Universal Robots URScript: move_path_1.script

def move_path_1():
  global _hidden_verificationVariable=0
  step_count_bb260f9f_b35d_4fa5_9196_51f97d34692a = 0.0
  thread Step_Counter_Thread_3f57fde8_be87_45f6_b73f_8ef8e3528eee():
    while (True):
      step_count_bb260f9f_b35d_4fa5_9196_51f97d34692a = step_count_bb260f9f_b35d_4fa5_9196_51f97d34692a + 1.0
      sync()
    end
  end
  run Step_Counter_Thread_3f57fde8_be87_45f6_b73f_8ef8e3528eee()
  set_gravity([0.0, 0.0, 9.82])
  set_standard_analog_input_domain(0, 1)
  set_standard_analog_input_domain(1, 1)
  set_tool_analog_input_domain(0, 1)
  set_tool_analog_input_domain(1, 1)
  set_analog_outputdomain(0, 0)
  set_analog_outputdomain(1, 0)
  set_input_actions_to_default()
  set_tcp(p[0.00855,-0.27152,0.102,1.2092,-1.2092,1.2092])
  set_target_payload(2.760000, [0.004000, -0.022000, 0.072000], [0.008360, 0.008360, 0.008360, 0.000000, 0.000000, 0.000000])
  set_safety_mode_transition_hardness(1)
  set_tool_communication(False, 115200, 0, 1, 1.5, 3.5)
  set_tool_output_mode(0)
  set_tool_digital_output_mode(0, 1)
  set_tool_digital_output_mode(1, 1)
  set_tool_voltage(0)
  global Plane_1=p[0.0,0.0,0.0,0.0,0.0,0.0]
  global Point_1=p[0.0,0.0,0.0,0.0,0.0,0.0]
  # begin: URCap Installation Node
  #   Source: MachineLogic for Universal Robots, 3.1.7, Vention Inc.
  #   Type: MachineLogic for Universal Robots
  def waitForResponse(expected_response_vention, cname_vention):
  response_vention = socket_read_string(cname_vention,timeout=15)
  while response_vention != expected_response_vention:
  sleep(0.01)
  response_vention = socket_read_string(cname_vention,timeout=15)
  end
  sleep(0.01)
  sync()
  end
  def sendString(string_vention, expected_response_vention, cname_vention):
  socket_send_string(str_cat(string_vention,";"), cname_vention)
  response_vention = socket_read_string(cname_vention,timeout=15)
  if(response_vention == "nAck"):
  popup("nAck received")
  end
  while response_vention != expected_response_vention:
  sleep(0.01)
  response_vention = socket_read_string(cname_vention,timeout=15)
  if(response_vention == "nAck"):
  popup("nAck received")
  end
  end
  sleep(0.01)
  sync()
  end
  def sendStringNAck(string_vention, expected_response_vention, cname_vention):
  socket_send_string(str_cat(string_vention,";"), cname_vention)
  response_vention = socket_read_string(cname_vention,timeout=15)
  if(response_vention == "nAck"):
  popup("nAck received")
  end
  while(response_vention != expected_response_vention and response_vention != "nAck"):
  sleep(0.01)
  response_vention = socket_read_string(cname_vention,timeout=15)
  if(response_vention == "nAck"):
  popup("nAck received",blocking=True)
  end
  end
  sleep(0.01)
  sync()
  end
  def sendStringWithTimeout(string_vention, expected_response_vention, cname_vention):
  socket_send_string(str_cat(string_vention,";"), cname_vention)
  response_vention = socket_read_string(cname_vention,timeout=10)
  if(response_vention == "nAck"):
  popup("nAck received"+string_vention)
  end
  sleep(0.01)
  sync()
  end
  def pollString(string_vention, expected_response_vention, cname_vention):
  socket_send_string(str_cat(string_vention,";"), cname_vention)
  response_vention = socket_read_string(cname_vention,timeout=15)
  if(response_vention == "nAck"):
  popup("nAck received")
  end
  while response_vention != expected_response_vention:
  sleep(1)
  socket_send_string(str_cat(string_vention,";"), cname_vention)
  response_vention = socket_read_string(cname_vention,timeout=15)
  if(response_vention == "nAck"):
  popup("nAck received")
  end
  end
  sleep(0.01)
  sync()
  end
  def sendVariable(var_vention, data_vention, expected_response_vention, cname_vention):
  socket_set_var(var_vention, data_vention, cname_vention)
  response_vention = socket_read_string(cname_vention,timeout=15)
  if(response_vention == "nAck"):
  popup("nAck received")
  end
  while response_vention != expected_response_vention:
  sleep(0.01)
  response_vention = socket_read_string(cname_vention,timeout=15)
  if(response_vention == "nAck"):
  popup("nAck received")
  end
  end
  sleep(0.01)
  sync()
  end
  def intToString(integer_vention,cname_vention):
  stringFix=""
  multiplier_vention123=1
  if integer_vention<0:
  stringFix="-"
  multiplier_vention123=-1
  end
  socket_set_var("GetString",integer_vention*multiplier_vention123,cname_vention)
  string_vention=""
  while string_vention=="":
  sleep(0.01)
  string_vention=socket_read_string(cname_vention,timeout=15)
  end
  sleep(0.01)
  sync()
  string_vention=stringFix+string_vention
  return string_vention
  end
  string_vention=""
  isVentionMovementBusy = False
  isVentionParallelMovementSendingScript = False
  ventionThreadHandle = 1
  isVentionMovementBusyMachineMotion1 = False
  isVentionParallelMovementSendingScriptMachineMotion1 = False
  socket_vention = socket_open("192.168.3.52", 9999, "MachineMotion1")
  if socket_vention==False:
  popup("Check configuration, can't connect to MachineMotion")
  end
  waitForResponse("MachineMotion connection established", "MachineMotion1")
  sendString("isReady", "MachineMotion isReady = true", "MachineMotion1")
  sendStringWithTimeout("setURCapVersion2", "setURCapVersion loaded", "MachineMotion1")
  sendString("SET speed_v2 1000000", "Ack", "MachineMotion1")
  sendString("SET acceleration_v2 100000", "Ack", "MachineMotion1")
  sendString("SET de_axis_1_microsteps_config 8", "Ack", "MachineMotion1")
  sendString("SET de_axis_1_mechanical_gain_config_v2 150000.0", "Ack", "MachineMotion1")
  sendString("SET de_axis_1_direction_config 1", "Ack", "MachineMotion1")
  sendString("SET de_axis_1_type_config Custom Actuator ", "Ack", "MachineMotion1")
  sendString("de_axis_1_config_exec", "Ack", "MachineMotion1")
  # end: URCap Installation Node
  global Waypoint_1_p=p[-.372860657265, .716170383118, .314676530127, 1.570809017190, -.000000152759, .000003968716]
  global Waypoint_1_q=[-1.3816140333758753, -1.0546258252910157, 1.8334205786334437, -0.7777959269336243, -1.3827489058123987, 6.28196907043457]
  while (True):
    $ 2 "Robot Program"
    $ 3 "pa1≔path1[1]"
    global pa1=path1[1]
    $ 4 "pa2≔path1[2]"
    global pa2=path1[2]
    $ 5 "p1≔path1[3]"
    global p1=path1[3]
    $ 6 "p2≔path1[4]"
    global p2=path1[4]
    $ 7 "p4≔path1[6]"
    global p4=path1[6]
    $ 8 "p5≔path1[7]"
    global p5=path1[7]
    $ 9 "pr1≔path1[8]"
    global pr1=path1[8]
    $ 10 "pvr1≔path1[12]"
    global pvr1=path1[12]
    $ 11 "pvr2≔path1[13]"
    global pvr2=path1[13]
    $ 12 "MoveJ"
    $ 13 "Waypoint_1" "breakAfter"
    movej(get_inverse_kin(Waypoint_1_p, qnear=Waypoint_1_q), a=1.3962634015954636, v=1.0471975511965976)
    $ 14 "MoveJ"
    $ 15 "pa1" "breakAfter"
    movej(pa1, a=1.3962634015954636, v=1.0471975511965976)
    $ 16 "MoveL"
    $ 17 "pa2" "breakAfter"
    movel(pa2, a=1.2, v=0.2)
    $ 18 "MoveL"
    $ 19 "p1" "breakAfter"
    movel(p1, a=1.2, v=0.05)
    $ 20 "Wait: 1.0"
    sleep(1.0)
    $ 21 "MoveP"
    $ 22 "p2" "breakAfter"
    movep(p2, a=1.2, v=0.012, r=0.025)
    $ 23 "Script: speedl_test2.script"
    #rot_speed=0.1
    #current_pose=get_actual_tcp_pose()
    #time_int = 5
    #target_pose=pose_trans(current_pose, p[0,0,0,0,0,rot_speed*time_int])
    #speedl(pose_sub(target_pose, current_pose), rot_speed, time_int)

    #get the headings and compare
    #current heading
    heading1=path1[9]
    #destination heading
    heading3 = path1[11]
    headingdelta = heading3 - heading1
    time_int = 3 #const
    rot_speed = headingdelta/time_int

    speedl([0,0,0,0,0,rot_speed],0.5,time_int)
    $ 24 "MoveP"
    $ 25 "p5" "breakAfter"
    movep(p5, a=1.2, v=0.012, r=0.025)
    $ 28 "MoveL"
    $ 29 "pr1" "breakAfter"
    movel(pr1, a=1.2, v=0.25)
    $ 30 "MoveJ"
    $ 31 "Waypoint_1" "breakAfter"
    movej(get_inverse_kin(Waypoint_1_p, qnear=Waypoint_1_q), a=1.3962634015954636, v=1.0471975511965976)
  end
end
